{attribute 'qualified_only'}
{attribute 'strict'}
TYPE E_Pwr :
(
	UNKNOWN:=0,
	ON,
	OFF,
	DONE
);
END_TYPE

(* stored: Version 1.1.0.1, ProductVersion 3.1.4022.12
   DUT E_Pwr: Id {a3e2778b-f5bd-457b-bebe-8a897a0948a4} *)
